INTERFACE ITF_Factory

METHOD Create : ITF_Cyclic
VAR_INPUT
END_VAR
END_METHOD

END_INTERFACE

(* stored: Version 1.1.0.1, ProductVersion 3.1.4024.12
   Itf ITF_Factory: Id {0c572baf-718a-40cb-be57-a4faab9984f5}
   Method Create: Id {07025c56-0565-495b-8006-364c8a17b066} *)
